FUNCTION_BLOCK SocketRecieveTask
VAR_INPUT
END_VAR
VAR_OUTPUT
END_VAR
VAR
END_VAR

END_FUNCTION_BLOCK

(* stored: Version 1.1.0.1, ProductVersion 3.1.4024.12
   POU SocketRecieveTask: Id {4c37506a-f01e-46ef-8308-65996d9f9557}, SpecialFunc None *)
